PROGRAM PRG_Calibration
VAR_OUTPUT
    bCalibrationFinished : BOOL;  // Indica o fim com sucesso da calibração
END_VAR
VAR
	
END_VAR

METHOD Reset : BOOL
VAR_INPUT
END_VAR
END_METHOD

END_PROGRAM

(* stored: Version 1.1.0.1, ProductVersion 3.1.4024.12
   POU PRG_Calibration: Id {f2ab8e02-eb8c-441d-b1b0-c2b3833b2b19}, SpecialFunc None
   Method Reset: Id {27813d8d-2df7-44d9-b974-4b44cba9f55d} *)
